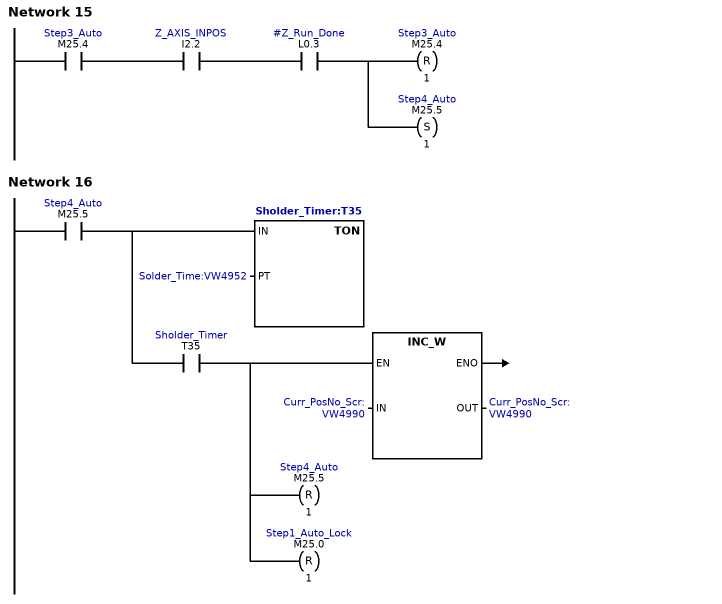
[picture p24: SBR34 networks 15-16]
Network 15
LD     Step3_Auto:M25.4
A      Z_AXIS_INPOS:I2.2
A      #Z_Run_Done:L0.3
R      Step3_Auto:M25.4, 1
S      Step4_Auto:M25.5, 1
Network 16
LD     Step4_Auto:M25.5
TON    Sholder_Timer:T35, Solder_Time:VW4952
A      Sholder_Timer:T35
INCW   Curr_PosNo_Scr:VW4990
R      Step4_Auto:M25.5, 1
R      Step1_Auto_Lock:M25.0, 1
END_SUBROUTINE_BLOCK

SUBROUTINE_BLOCK Setting:SBR35
TITLE=子例程注释
VAR_INPUT
MainScreen:WORD;	// LW0 
END_VAR
VAR
X_Home_Err:BYTE;	// LB2 
Y_Home_Err:BYTE;	// LB3 
Z_Home_Err:BYTE;	// LB4 
X_Teach_Done:BOOL;	// L5.0 
Y_Teach_Done:BOOL;	// L5.1 
Z_Teach_Done:BOOL;	// L5.2 
Z_Up_Done:BOOL;	// L5.3 
X_JOG_ERR:BYTE;	// LB6 
Y_JOG_ERR:BYTE;	// LB7 
Z_JOG_ERR:BYTE;	// LB8 
X_Curr_Dir:BOOL;	// L9.0 
Y_Curr_Dir:BOOL;	// L9.1 
Z_Curr_Dir:BOOL;	// L9.2 
END_VAR
BEGIN
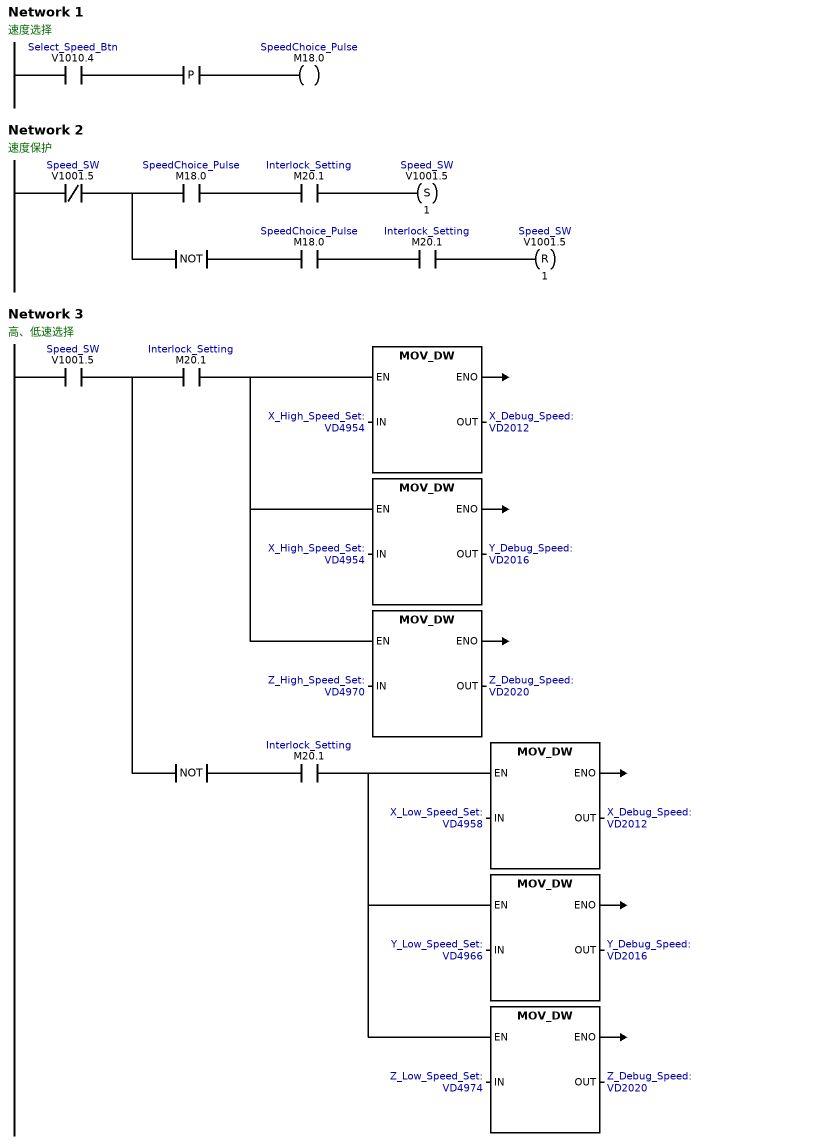
Network 1
// 速度选择
LD     Select_Speed_Btn:V1010.4
EU
=      SpeedChoice_Pulse:M18.0
Network 2
// 速度保护
LDN    Speed_SW:V1001.5
LPS
A      SpeedChoice_Pulse:M18.0
A      Interlock_Setting:M20.1
S      Speed_SW:V1001.5, 1
LPP
NOT
A      SpeedChoice_Pulse:M18.0
A      Interlock_Setting:M20.1
R      Speed_SW:V1001.5, 1
Network 3
// 高、低速选择
LD     Speed_SW:V1001.5
LPS
A      Interlock_Setting:M20.1
MOVD   X_High_Speed_Set:VD4954, X_Debug_Speed:VD2012
MOVD   X_High_Speed_Set:VD4954, Y_Debug_Speed:VD2016
MOVD   Z_High_Speed_Set:VD4970, Z_Debug_Speed:VD2020
LPP
NOT
A      Interlock_Setting:M20.1
MOVD   X_Low_Speed_Set:VD4958, X_Debug_Speed:VD2012
MOVD   Y_Low_Speed_Set:VD4966, Y_Debug_Speed:VD2016
MOVD   Z_Low_Speed_Set:VD4974, Z_Debug_Speed:VD2020
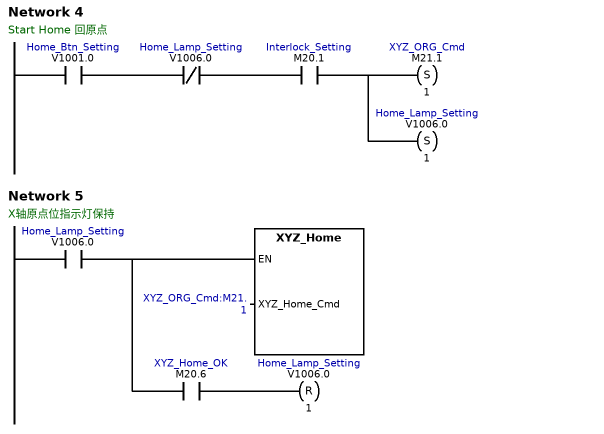
Network 4
// Start Home 回原点
LD     Home_Btn_Setting:V1001.0
AN     Home_Lamp_Setting:V1006.0
A      Interlock_Setting:M20.1
S      XYZ_ORG_Cmd:M21.1, 1
S      Home_Lamp_Setting:V1006.0, 1
Network 5
// X轴原点位指示灯保持
LD     Home_Lamp_Setting:V1006.0
CALL   XYZ_Home:SBR37, XYZ_ORG_Cmd:M21.1
A      XYZ_Home_OK:M20.6
R      Home_Lamp_Setting:V1006.0, 1
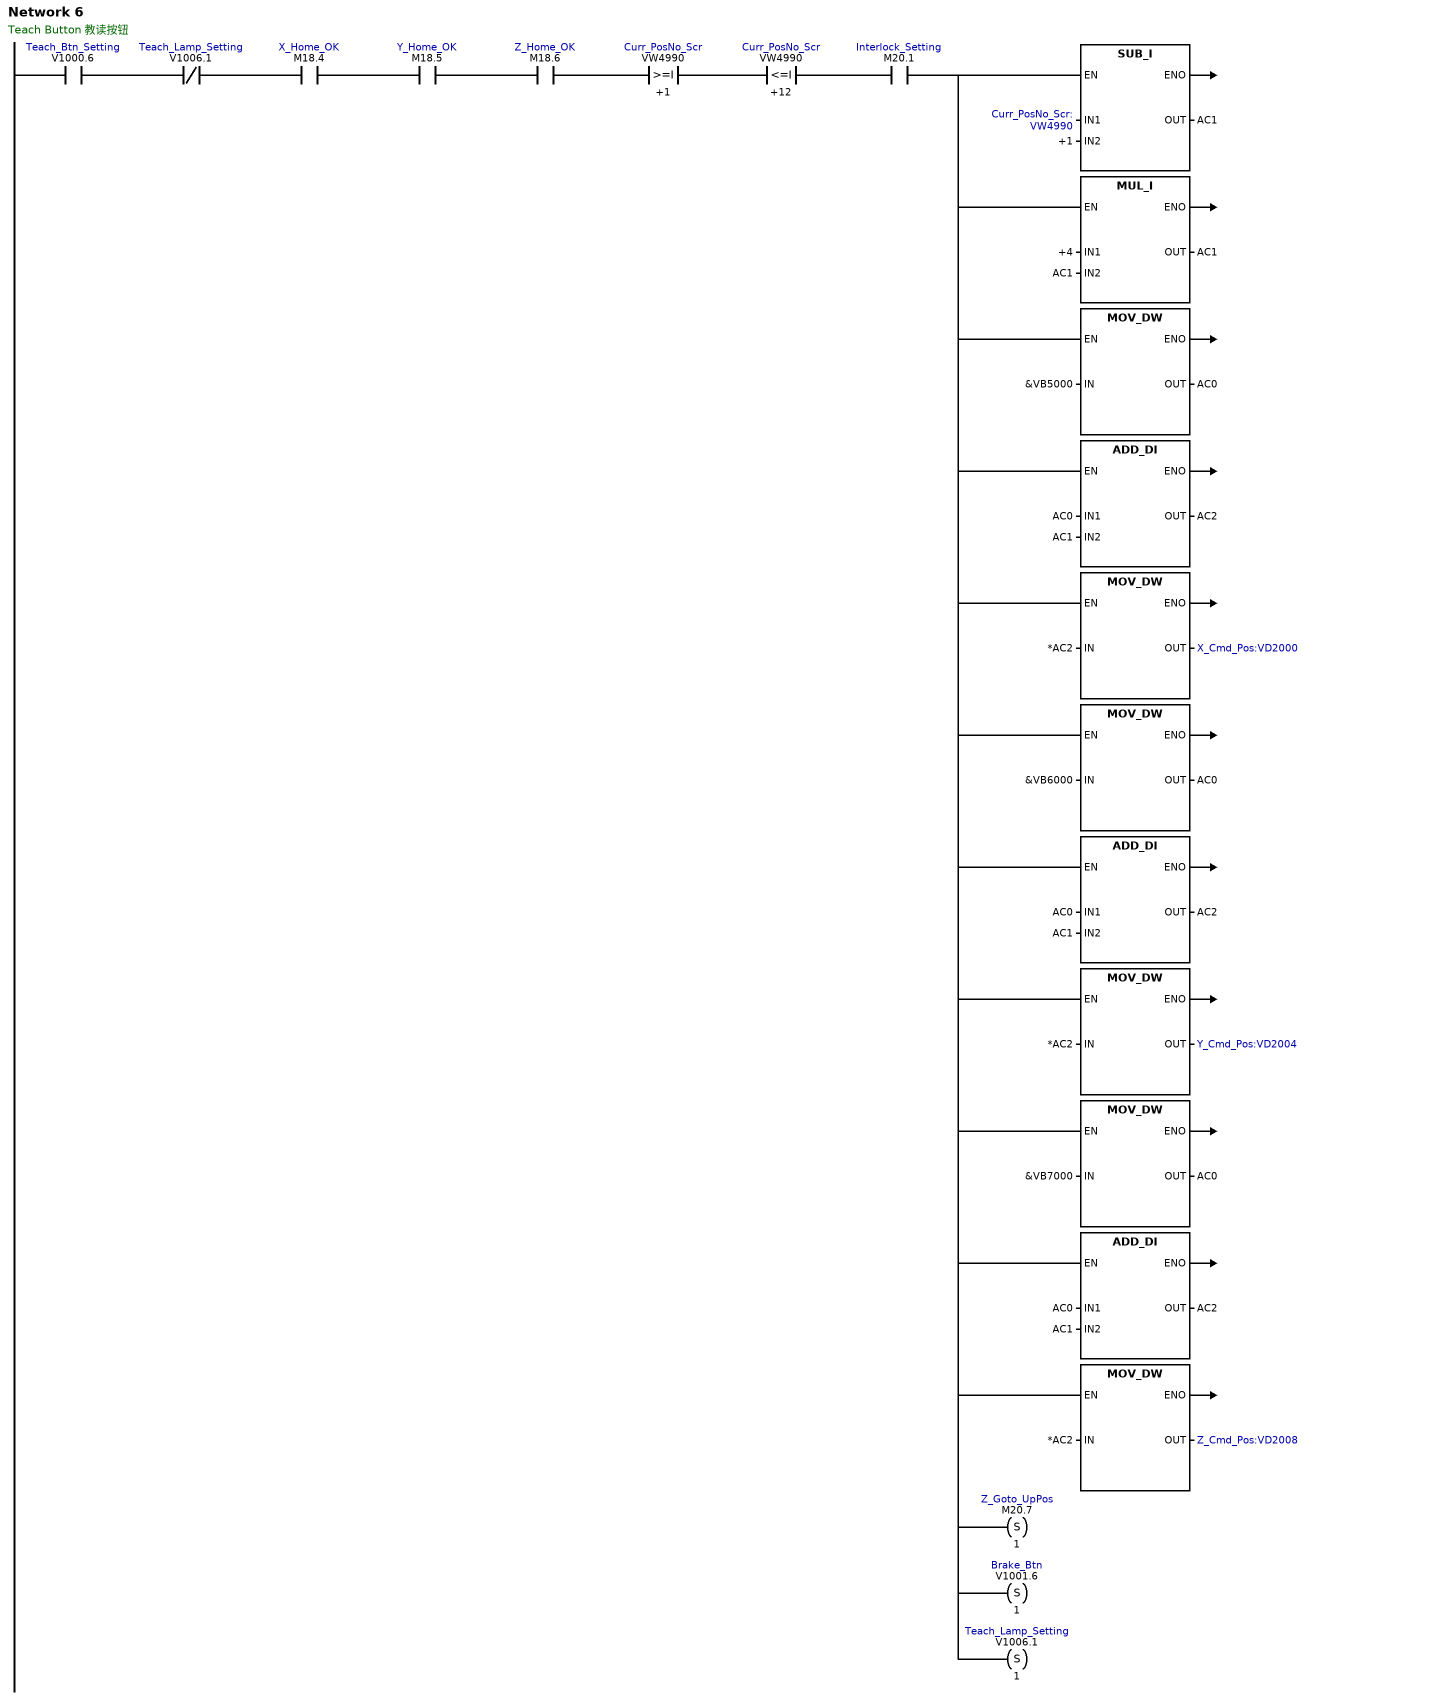
Network 6
// Teach Button 教读按钮 
LD     Teach_Btn_Setting:V1000.6
AN     Teach_Lamp_Setting:V1006.1
A      X_Home_OK:M18.4
A      Y_Home_OK:M18.5
A      Z_Home_OK:M18.6
AW>=   Curr_PosNo_Scr:VW4990, +1
AW<=   Curr_PosNo_Scr:VW4990, +12
A      Interlock_Setting:M20.1
MOVW   Curr_PosNo_Scr:VW4990, AC1
-I     +1, AC1
*I     +4, AC1
MOVD   &VB5000, AC0
MOVD   AC0, AC2
+D     AC1, AC2
MOVD   *AC2, X_Cmd_Pos:VD2000
MOVD   &VB6000, AC0
MOVD   AC0, AC2
+D     AC1, AC2
MOVD   *AC2, Y_Cmd_Pos:VD2004
MOVD   &VB7000, AC0
MOVD   AC0, AC2
+D     AC1, AC2
MOVD   *AC2, Z_Cmd_Pos:VD2008
S      Z_Goto_UpPos:M20.7, 1
S      Brake_Btn:V1001.6, 1
S      Teach_Lamp_Setting:V1006.1, 1
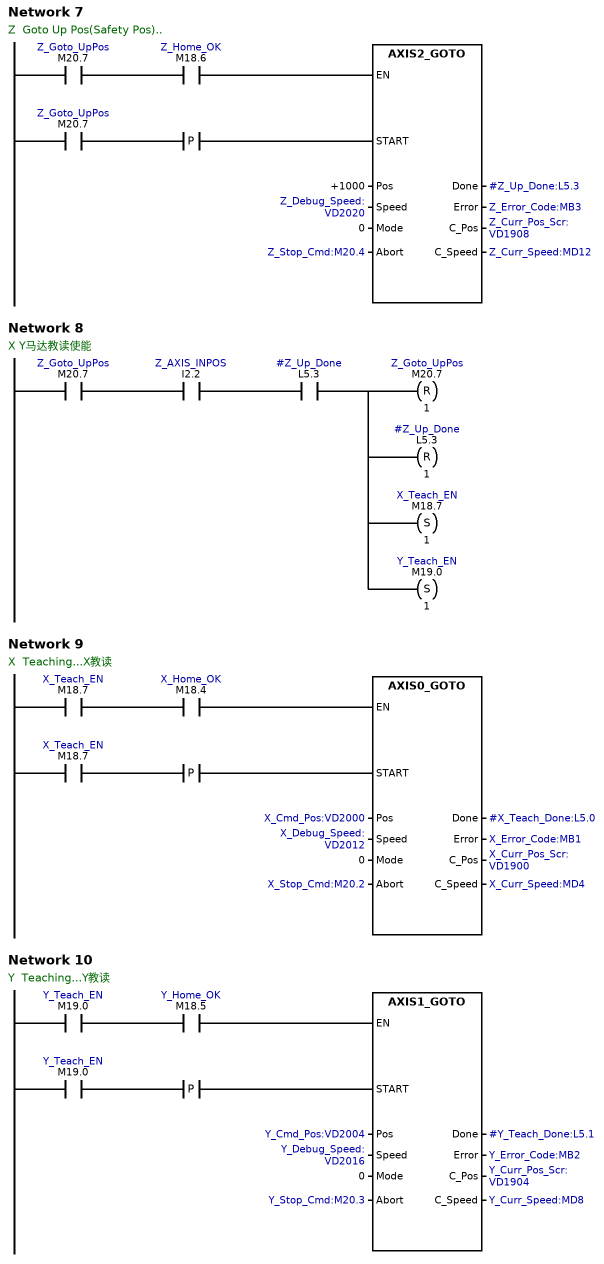
Network 7
// Z  Goto Up Pos(Safety Pos)..
LD     Z_Goto_UpPos:M20.7
A      Z_Home_OK:M18.6
=      L60.0
LD     Z_Goto_UpPos:M20.7
EU
=      L63.7
LD     L60.0
CALL   AXIS2_GOTO:SBR25, L63.7, +1000, Z_Debug_Speed:VD2020, 0, Z_Stop_Cmd:M20.4, #Z_Up_Done:L5.3, Z_Error_Code:MB3, Z_Curr_Pos_Scr:VD1908, Z_Curr_Speed:MD12
Network 8
// X Y马达教读使能
LD     Z_Goto_UpPos:M20.7
A      Z_AXIS_INPOS:I2.2
A      #Z_Up_Done:L5.3
R      Z_Goto_UpPos:M20.7, 1
R      #Z_Up_Done:L5.3, 1
S      X_Teach_EN:M18.7, 1
S      Y_Teach_EN:M19.0, 1
Network 9
// X  Teaching...X教读
LD     X_Teach_EN:M18.7
A      X_Home_OK:M18.4
=      L60.0
LD     X_Teach_EN:M18.7
EU
=      L63.7
LD     L60.0
CALL   AXIS0_GOTO:SBR3, L63.7, X_Cmd_Pos:VD2000, X_Debug_Speed:VD2012, 0, X_Stop_Cmd:M20.2, #X_Teach_Done:L5.0, X_Error_Code:MB1, X_Curr_Pos_Scr:VD1900, X_Curr_Speed:MD4
Network 10
// Y  Teaching...Y教读
LD     Y_Teach_EN:M19.0
A      Y_Home_OK:M18.5
=      L60.0
LD     Y_Teach_EN:M19.0
EU
=      L63.7
LD     L60.0
CALL   AXIS1_GOTO:SBR14, L63.7, Y_Cmd_Pos:VD2004, Y_Debug_Speed:VD2016, 0, Y_Stop_Cmd:M20.3, #Y_Teach_Done:L5.1, Y_Error_Code:MB2, Y_Curr_Pos_Scr:VD1904, Y_Curr_Speed:MD8
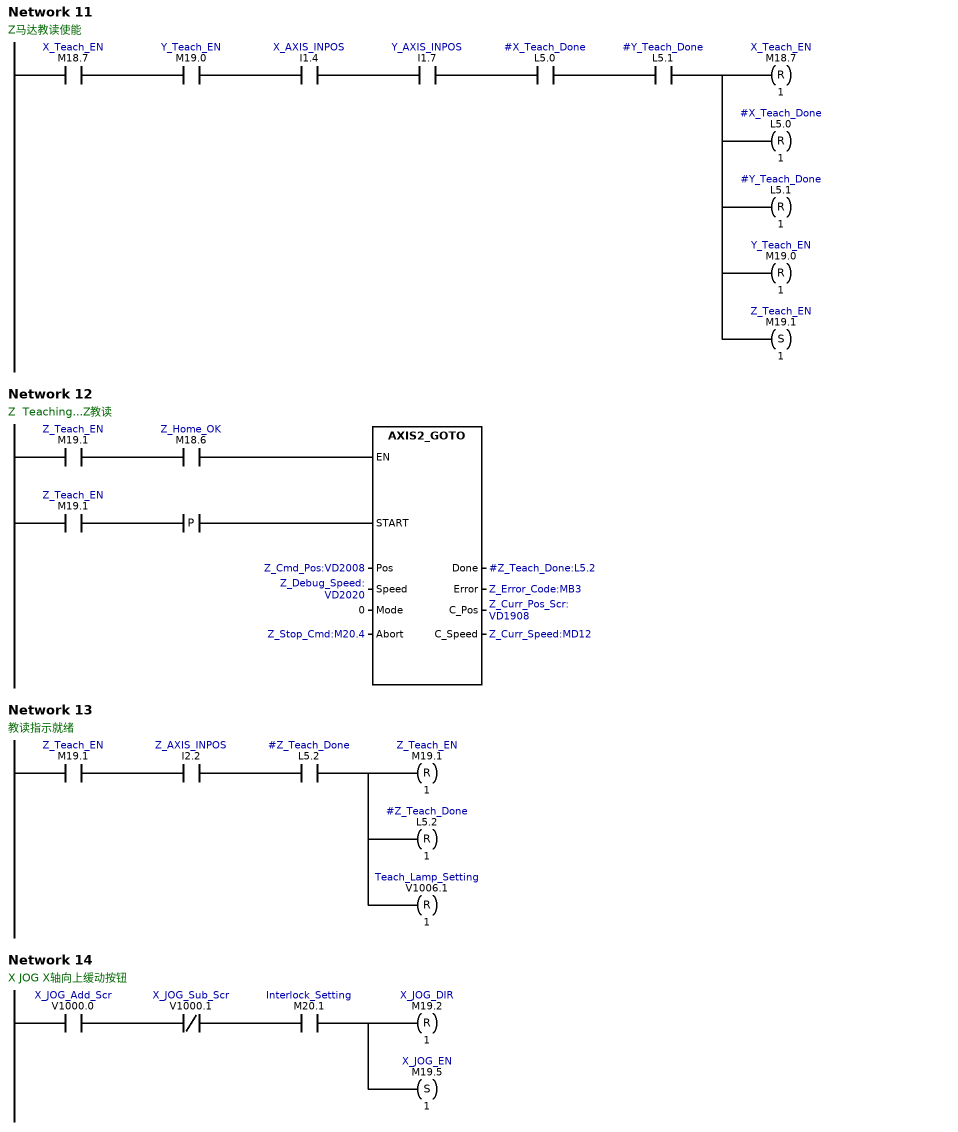
Network 11
// Z马达教读使能
LD     X_Teach_EN:M18.7
A      Y_Teach_EN:M19.0
A      X_AXIS_INPOS:I1.4
A      Y_AXIS_INPOS:I1.7
A      #X_Teach_Done:L5.0
A      #Y_Teach_Done:L5.1
R      X_Teach_EN:M18.7, 1
R      #X_Teach_Done:L5.0, 1
R      #Y_Teach_Done:L5.1, 1
R      Y_Teach_EN:M19.0, 1
S      Z_Teach_EN:M19.1, 1
Network 12
// Z  Teaching...Z教读
LD     Z_Teach_EN:M19.1
A      Z_Home_OK:M18.6
=      L60.0
LD     Z_Teach_EN:M19.1
EU
=      L63.7
LD     L60.0
CALL   AXIS2_GOTO:SBR25, L63.7, Z_Cmd_Pos:VD2008, Z_Debug_Speed:VD2020, 0, Z_Stop_Cmd:M20.4, #Z_Teach_Done:L5.2, Z_Error_Code:MB3, Z_Curr_Pos_Scr:VD1908, Z_Curr_Speed:MD12
Network 13
// 教读指示就绪
LD     Z_Teach_EN:M19.1
A      Z_AXIS_INPOS:I2.2
A      #Z_Teach_Done:L5.2
R      Z_Teach_EN:M19.1, 1
R      #Z_Teach_Done:L5.2, 1
R      Teach_Lamp_Setting:V1006.1, 1
Network 14
// X JOG X轴向上缓动按钮
LD     X_JOG_Add_Scr:V1000.0
AN     X_JOG_Sub_Scr:V1000.1
A      Interlock_Setting:M20.1
R      X_JOG_DIR:M19.2, 1
S      X_JOG_EN:M19.5, 1
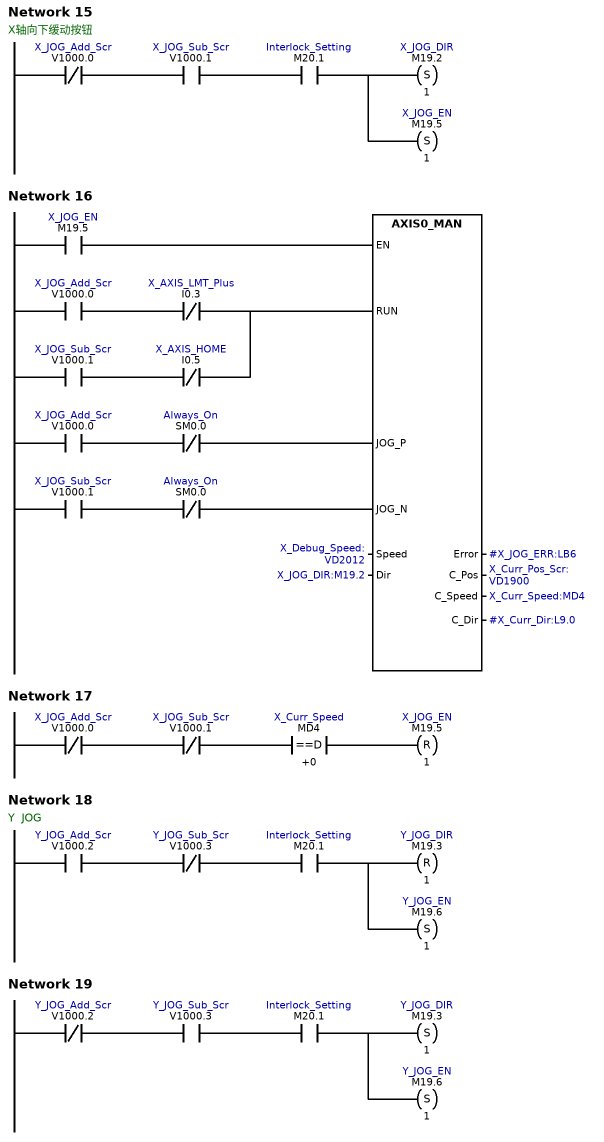
Network 15
// X轴向下缓动按钮
LDN    X_JOG_Add_Scr:V1000.0
A      X_JOG_Sub_Scr:V1000.1
A      Interlock_Setting:M20.1
S      X_JOG_DIR:M19.2, 1
S      X_JOG_EN:M19.5, 1
Network 16
LD     X_JOG_EN:M19.5
=      L60.0
LD     X_JOG_Add_Scr:V1000.0
AN     X_AXIS_LMT_Plus:I0.3
LD     X_JOG_Sub_Scr:V1000.1
AN     X_AXIS_HOME:I0.5
OLD
=      L63.7
LD     X_JOG_Add_Scr:V1000.0
AN     Always_On:SM0.0
=      L63.6
LD     X_JOG_Sub_Scr:V1000.1
AN     Always_On:SM0.0
=      L63.5
LD     L60.0
CALL   AXIS0_MAN:SBR2, L63.7, L63.6, L63.5, X_Debug_Speed:VD2012, X_JOG_DIR:M19.2, #X_JOG_ERR:LB6, X_Curr_Pos_Scr:VD1900, X_Curr_Speed:MD4, #X_Curr_Dir:L9.0
Network 17
LDN    X_JOG_Add_Scr:V1000.0
AN     X_JOG_Sub_Scr:V1000.1
AD=    X_Curr_Speed:MD4, +0
R      X_JOG_EN:M19.5, 1
Network 18
// Y  JOG
LD     Y_JOG_Add_Scr:V1000.2
AN     Y_JOG_Sub_Scr:V1000.3
A      Interlock_Setting:M20.1
R      Y_JOG_DIR:M19.3, 1
S      Y_JOG_EN:M19.6, 1
Network 19
LDN    Y_JOG_Add_Scr:V1000.2
A      Y_JOG_Sub_Scr:V1000.3
A      Interlock_Setting:M20.1
S      Y_JOG_DIR:M19.3, 1
S      Y_JOG_EN:M19.6, 1
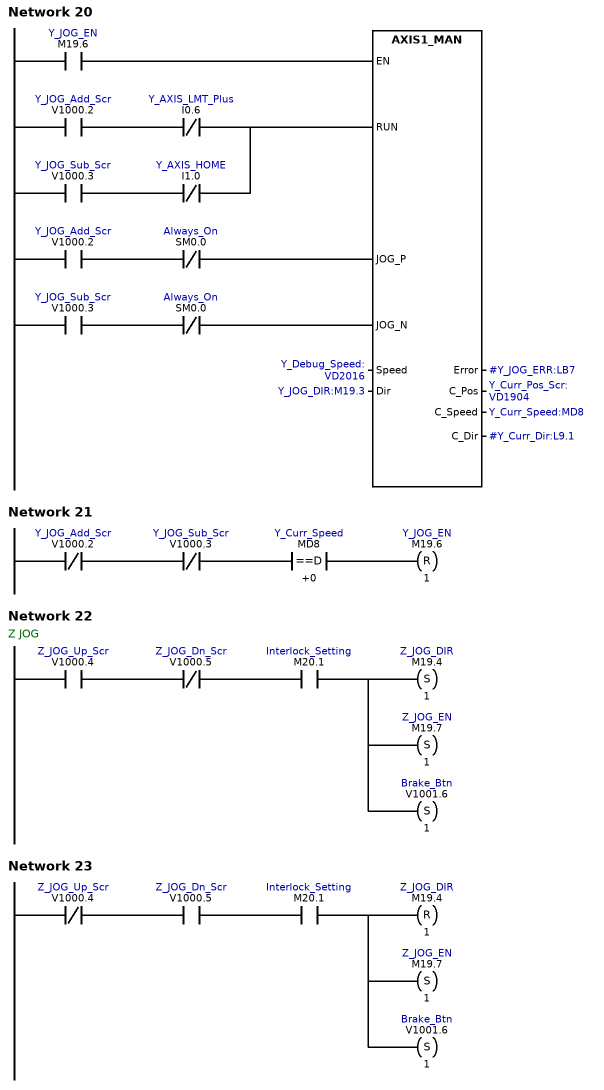
Network 20
LD     Y_JOG_EN:M19.6
=      L60.0
LD     Y_JOG_Add_Scr:V1000.2
AN     Y_AXIS_LMT_Plus:I0.6
LD     Y_JOG_Sub_Scr:V1000.3
AN     Y_AXIS_HOME:I1.0
OLD
=      L63.7
LD     Y_JOG_Add_Scr:V1000.2
AN     Always_On:SM0.0
=      L63.6
LD     Y_JOG_Sub_Scr:V1000.3
AN     Always_On:SM0.0
=      L63.5
LD     L60.0
CALL   AXIS1_MAN:SBR13, L63.7, L63.6, L63.5, Y_Debug_Speed:VD2016, Y_JOG_DIR:M19.3, #Y_JOG_ERR:LB7, Y_Curr_Pos_Scr:VD1904, Y_Curr_Speed:MD8, #Y_Curr_Dir:L9.1
Network 21
LDN    Y_JOG_Add_Scr:V1000.2
AN     Y_JOG_Sub_Scr:V1000.3
AD=    Y_Curr_Speed:MD8, +0
R      Y_JOG_EN:M19.6, 1
Network 22
// Z JOG
LD     Z_JOG_Up_Scr:V1000.4
AN     Z_JOG_Dn_Scr:V1000.5
A      Interlock_Setting:M20.1
S      Z_JOG_DIR:M19.4, 1
S      Z_JOG_EN:M19.7, 1
S      Brake_Btn:V1001.6, 1
Network 23
LDN    Z_JOG_Up_Scr:V1000.4
A      Z_JOG_Dn_Scr:V1000.5
A      Interlock_Setting:M20.1
R      Z_JOG_DIR:M19.4, 1
S      Z_JOG_EN:M19.7, 1
S      Brake_Btn:V1001.6, 1
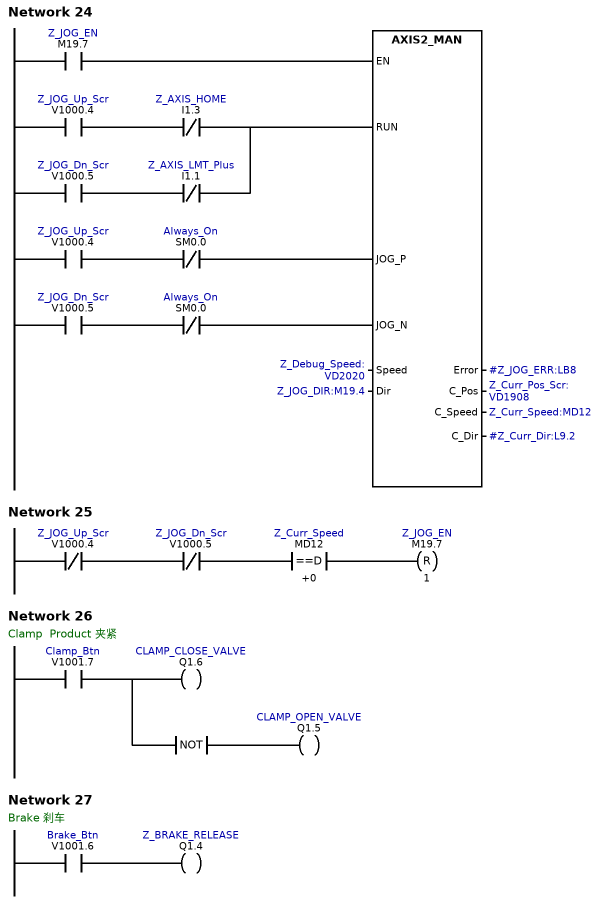
Network 24
LD     Z_JOG_EN:M19.7
=      L60.0
LD     Z_JOG_Up_Scr:V1000.4
AN     Z_AXIS_HOME:I1.3
LD     Z_JOG_Dn_Scr:V1000.5
AN     Z_AXIS_LMT_Plus:I1.1
OLD
=      L63.7
LD     Z_JOG_Up_Scr:V1000.4
AN     Always_On:SM0.0
=      L63.6
LD     Z_JOG_Dn_Scr:V1000.5
AN     Always_On:SM0.0
=      L63.5
LD     L60.0
CALL   AXIS2_MAN:SBR24, L63.7, L63.6, L63.5, Z_Debug_Speed:VD2020, Z_JOG_DIR:M19.4, #Z_JOG_ERR:LB8, Z_Curr_Pos_Scr:VD1908, Z_Curr_Speed:MD12, #Z_Curr_Dir:L9.2
Network 25
LDN    Z_JOG_Up_Scr:V1000.4
AN     Z_JOG_Dn_Scr:V1000.5
AD=    Z_Curr_Speed:MD12, +0
R      Z_JOG_EN:M19.7, 1
Network 26
// Clamp  Product 夹紧
LD     Clamp_Btn:V1001.7
=      CLAMP_CLOSE_VALVE:Q1.6
NOT
=      CLAMP_OPEN_VALVE:Q1.5
Network 27
// Brake 刹车
LD     Brake_Btn:V1001.6
=      Z_BRAKE_RELEASE:Q1.4
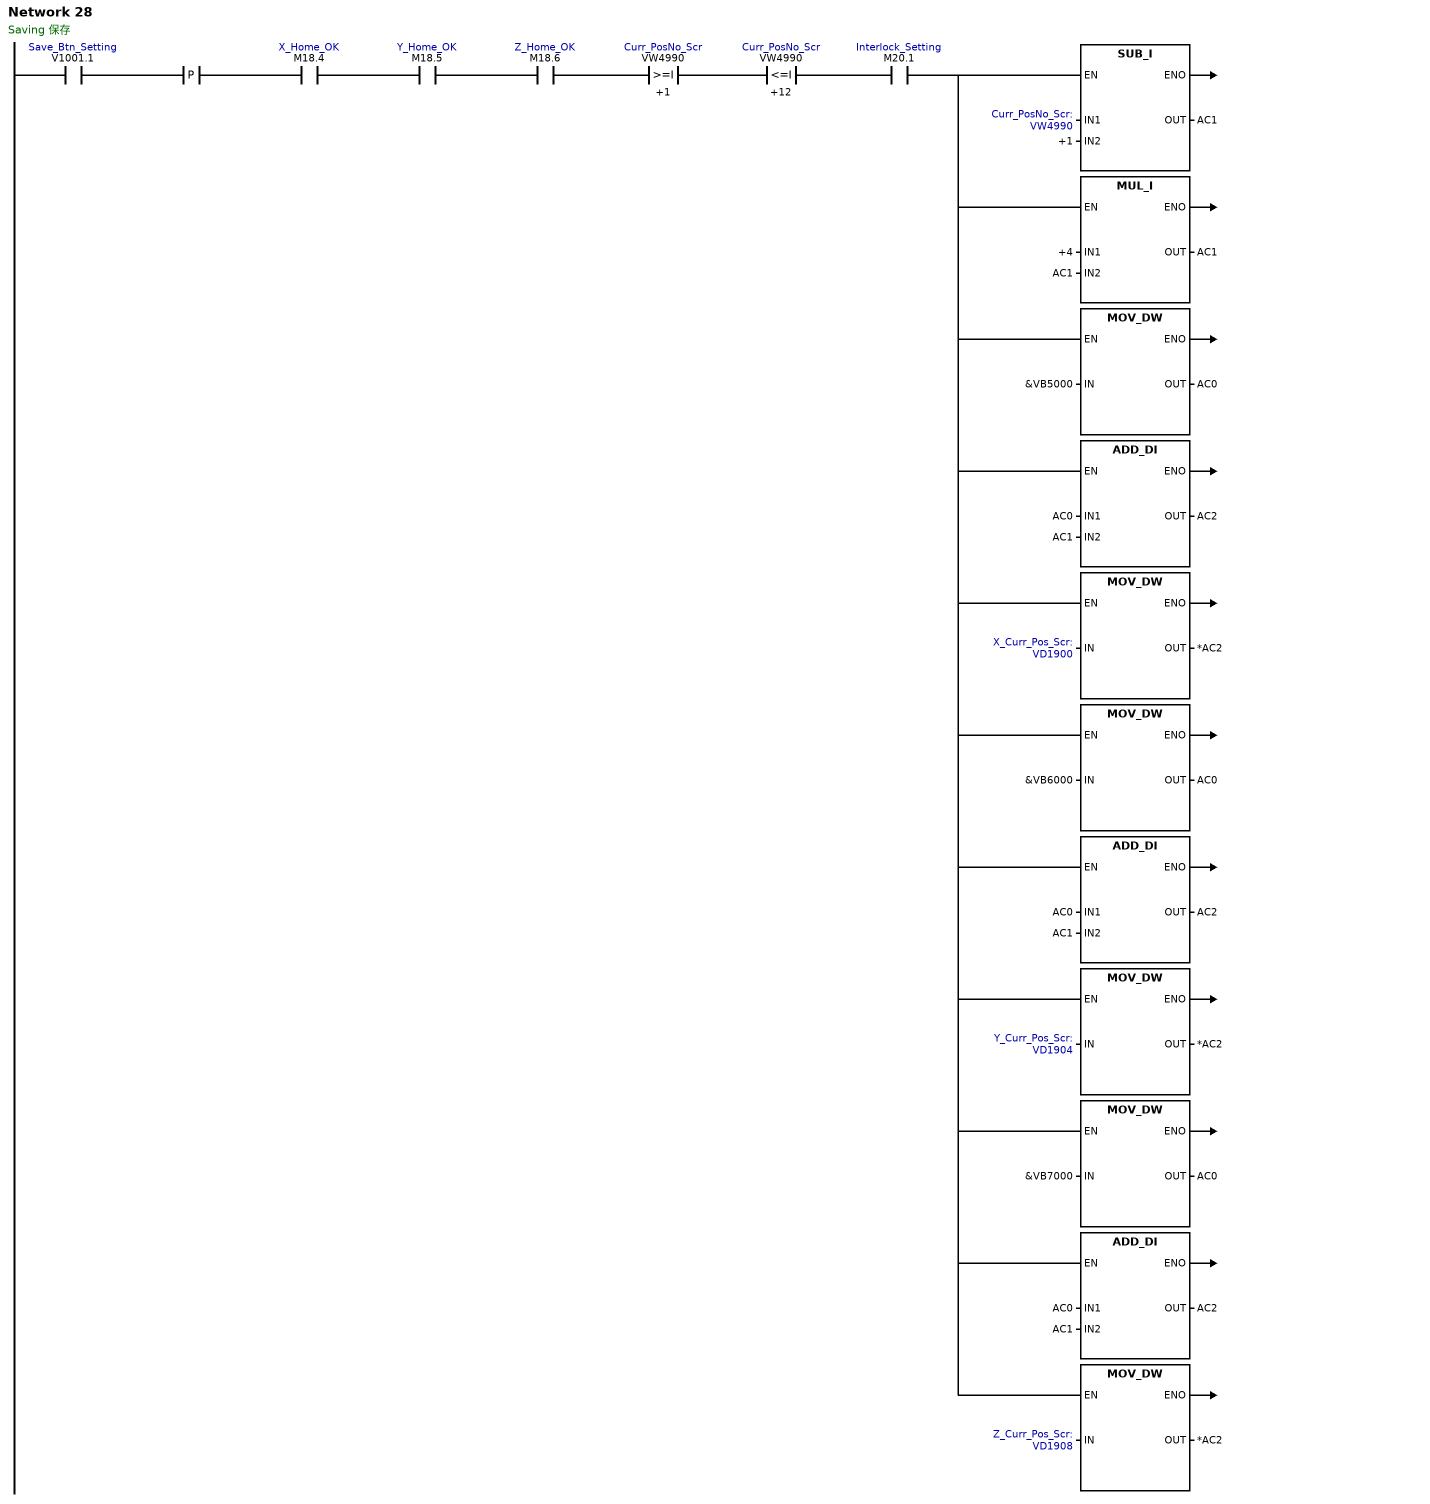
Network 28
// Saving 保存
LD     Save_Btn_Setting:V1001.1
EU
A      X_Home_OK:M18.4
A      Y_Home_OK:M18.5
A      Z_Home_OK:M18.6
AW>=   Curr_PosNo_Scr:VW4990, +1
AW<=   Curr_PosNo_Scr:VW4990, +12
A      Interlock_Setting:M20.1
MOVW   Curr_PosNo_Scr:VW4990, AC1
-I     +1, AC1
*I     +4, AC1
MOVD   &VB5000, AC0
MOVD   AC0, AC2
+D     AC1, AC2
MOVD   X_Curr_Pos_Scr:VD1900, *AC2
MOVD   &VB6000, AC0
MOVD   AC0, AC2
+D     AC1, AC2
MOVD   Y_Curr_Pos_Scr:VD1904, *AC2
MOVD   &VB7000, AC0
MOVD   AC0, AC2
+D     AC1, AC2
MOVD   Z_Curr_Pos_Scr:VD1908, *AC2
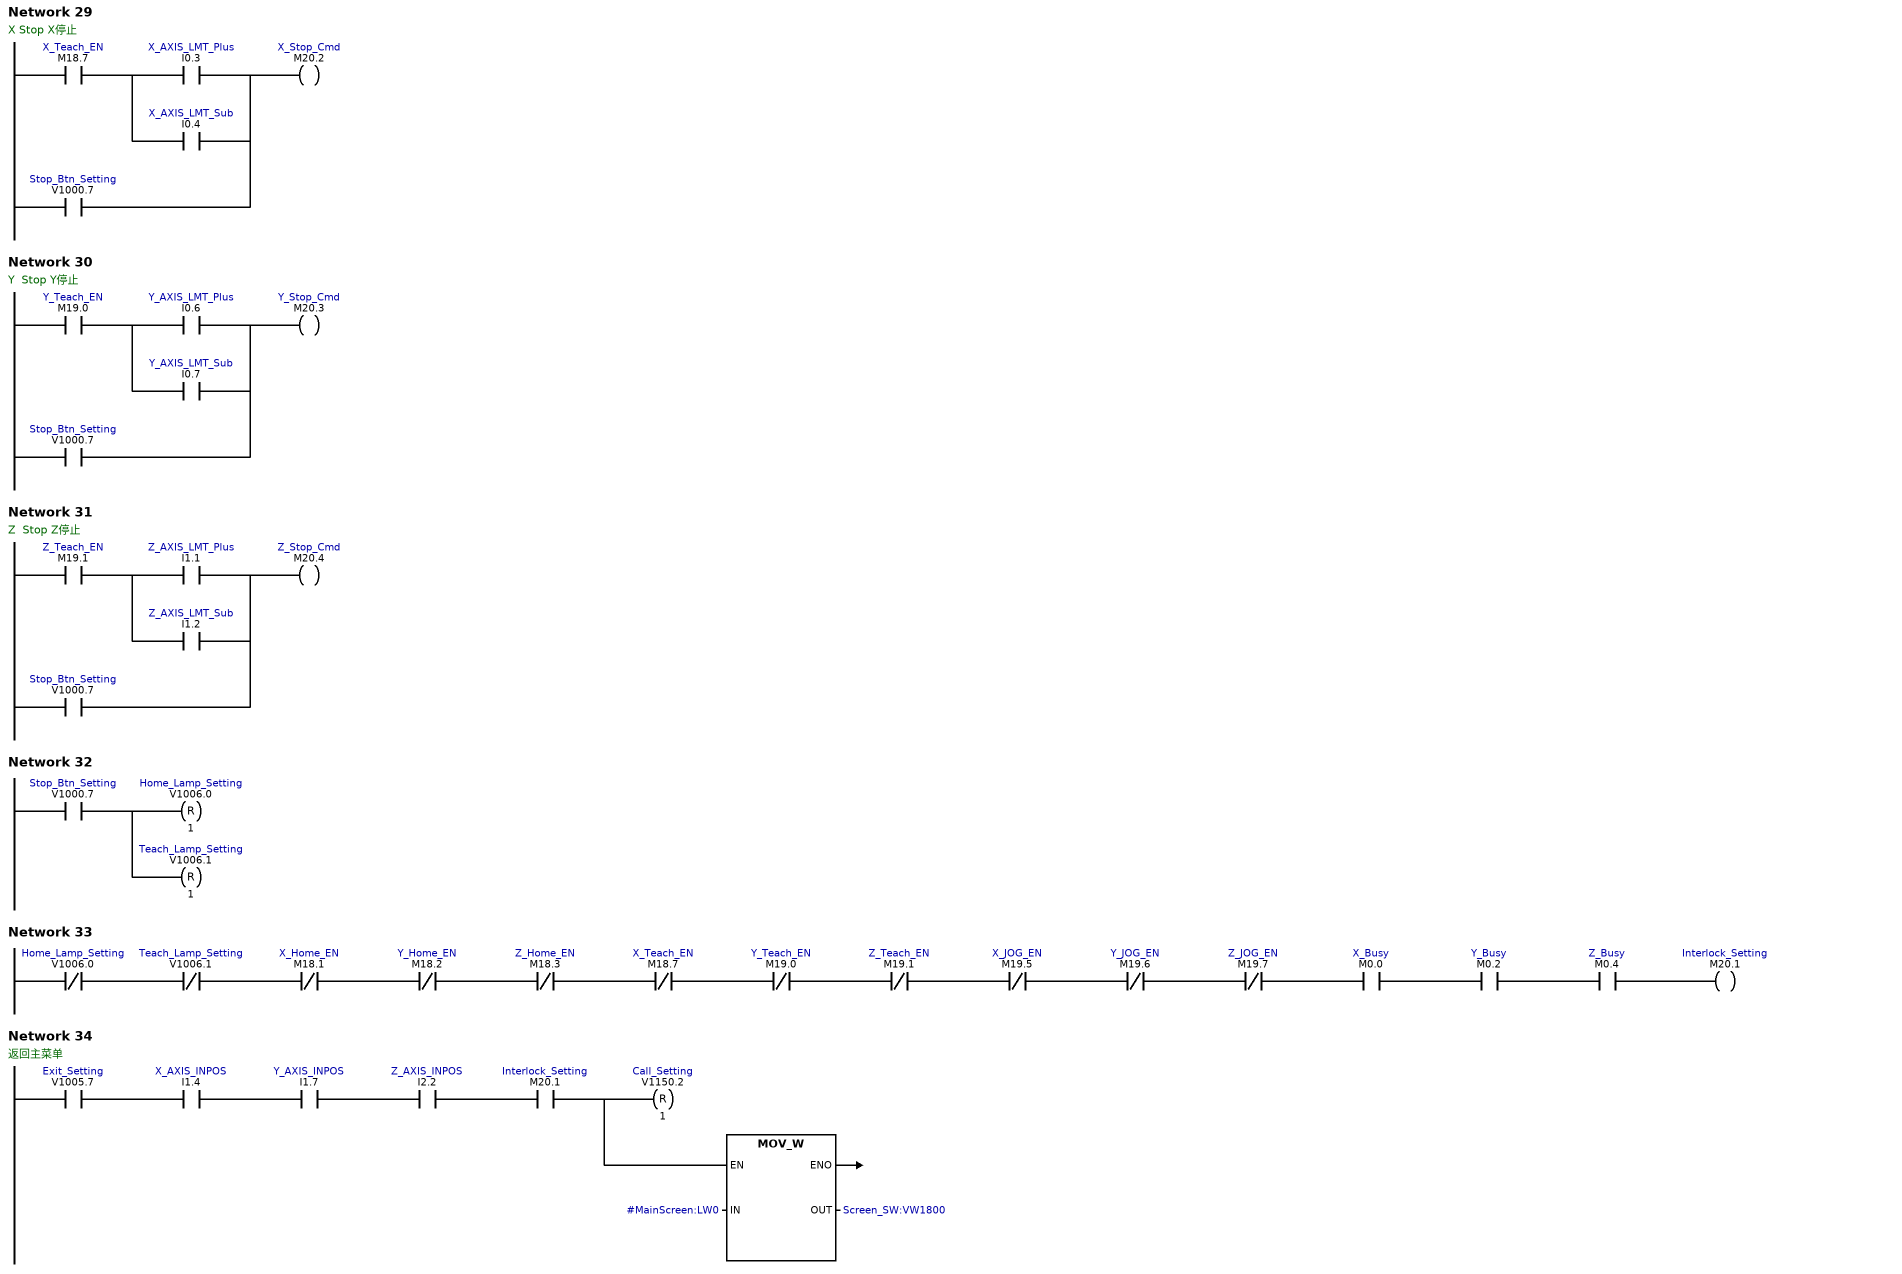
Network 29
// X Stop X停止
LD     X_Teach_EN:M18.7
LD     X_AXIS_LMT_Plus:I0.3
O      X_AXIS_LMT_Sub:I0.4
ALD
O      Stop_Btn_Setting:V1000.7
=      X_Stop_Cmd:M20.2
Network 30
// Y  Stop Y停止
LD     Y_Teach_EN:M19.0
LD     Y_AXIS_LMT_Plus:I0.6
O      Y_AXIS_LMT_Sub:I0.7
ALD
O      Stop_Btn_Setting:V1000.7
=      Y_Stop_Cmd:M20.3
Network 31
// Z  Stop Z停止
LD     Z_Teach_EN:M19.1
LD     Z_AXIS_LMT_Plus:I1.1
O      Z_AXIS_LMT_Sub:I1.2
ALD
O      Stop_Btn_Setting:V1000.7
=      Z_Stop_Cmd:M20.4
Network 32
LD     Stop_Btn_Setting:V1000.7
R      Home_Lamp_Setting:V1006.0, 1
R      Teach_Lamp_Setting:V1006.1, 1
Network 33
LDN    Home_Lamp_Setting:V1006.0
AN     Teach_Lamp_Setting:V1006.1
AN     X_Home_EN:M18.1
AN     Y_Home_EN:M18.2
AN     Z_Home_EN:M18.3
AN     X_Teach_EN:M18.7
AN     Y_Teach_EN:M19.0
AN     Z_Teach_EN:M19.1
AN     X_JOG_EN:M19.5
AN     Y_JOG_EN:M19.6
AN     Z_JOG_EN:M19.7
A      X_Busy:M0.0
A      Y_Busy:M0.2
A      Z_Busy:M0.4
=      Interlock_Setting:M20.1
Network 34
// 返回主菜单
LD     Exit_Setting:V1005.7
A      X_AXIS_INPOS:I1.4
A      Y_AXIS_INPOS:I1.7
A      Z_AXIS_INPOS:I2.2
A      Interlock_Setting:M20.1
R      Call_Setting:V1150.2, 1
MOVW   #MainScreen:LW0, Screen_SW:VW1800
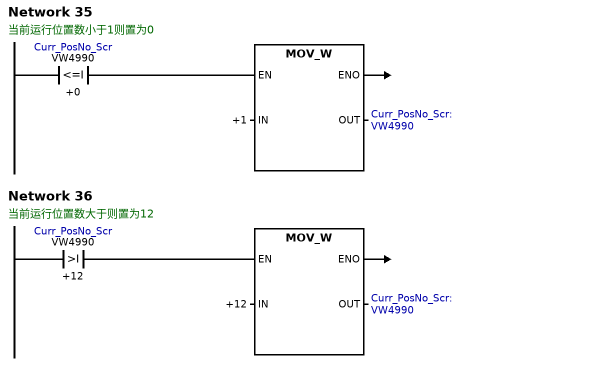
Network 35
// 当前运行位置数小于1则置为0
LDW<=  Curr_PosNo_Scr:VW4990, +0
MOVW   +1, Curr_PosNo_Scr:VW4990
Network 36
// 当前运行位置数大于则置为12
LDW>   Curr_PosNo_Scr:VW4990, +12
MOVW   +12, Curr_PosNo_Scr:VW4990
END_SUBROUTINE_BLOCK

SUBROUTINE_BLOCK Alarm_Process:SBR36
TITLE=子例程注释
BEGIN
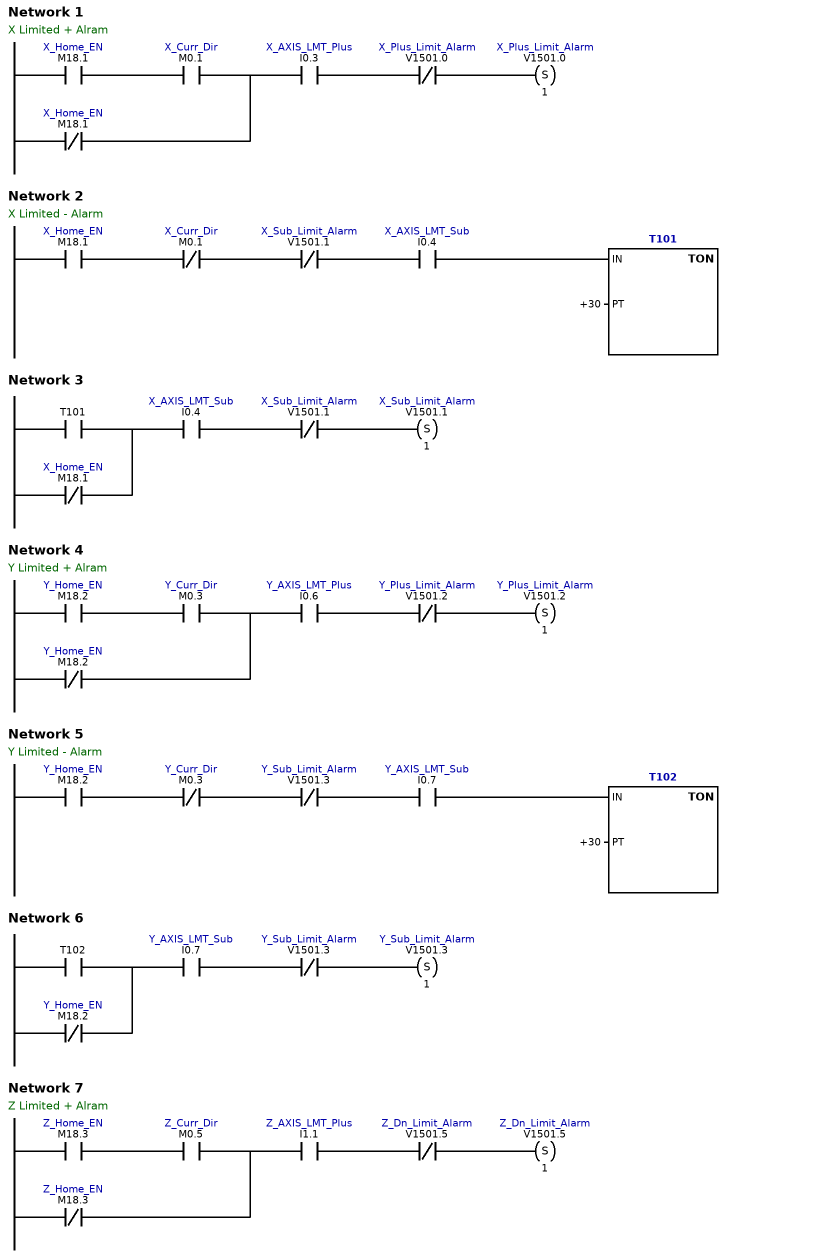
Network 1
// X Limited + Alram
LD     X_Home_EN:M18.1
A      X_Curr_Dir:M0.1
ON     X_Home_EN:M18.1
A      X_AXIS_LMT_Plus:I0.3
AN     X_Plus_Limit_Alarm:V1501.0
S      X_Plus_Limit_Alarm:V1501.0, 1
Network 2
// X Limited - Alarm
LD     X_Home_EN:M18.1
AN     X_Curr_Dir:M0.1
AN     X_Sub_Limit_Alarm:V1501.1
A      X_AXIS_LMT_Sub:I0.4
TON    T101, +30
Network 3
LD     T101
ON     X_Home_EN:M18.1
A      X_AXIS_LMT_Sub:I0.4
AN     X_Sub_Limit_Alarm:V1501.1
S      X_Sub_Limit_Alarm:V1501.1, 1
Network 4
// Y Limited + Alram
LD     Y_Home_EN:M18.2
A      Y_Curr_Dir:M0.3
ON     Y_Home_EN:M18.2
A      Y_AXIS_LMT_Plus:I0.6
AN     Y_Plus_Limit_Alarm:V1501.2
S      Y_Plus_Limit_Alarm:V1501.2, 1
Network 5
// Y Limited - Alarm
LD     Y_Home_EN:M18.2
AN     Y_Curr_Dir:M0.3
AN     Y_Sub_Limit_Alarm:V1501.3
A      Y_AXIS_LMT_Sub:I0.7
TON    T102, +30
Network 6
LD     T102
ON     Y_Home_EN:M18.2
A      Y_AXIS_LMT_Sub:I0.7
AN     Y_Sub_Limit_Alarm:V1501.3
S      Y_Sub_Limit_Alarm:V1501.3, 1
Network 7
// Z Limited + Alram
LD     Z_Home_EN:M18.3
A      Z_Curr_Dir:M0.5
ON     Z_Home_EN:M18.3
A      Z_AXIS_LMT_Plus:I1.1
AN     Z_Dn_Limit_Alarm:V1501.5
S      Z_Dn_Limit_Alarm:V1501.5, 1
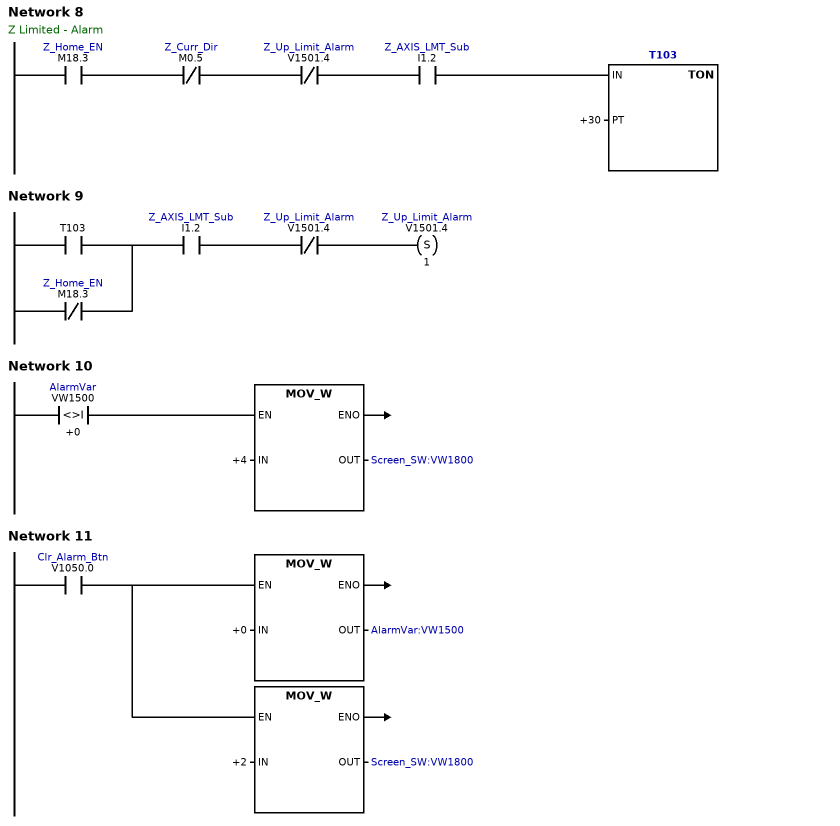
Network 8
// Z Limited - Alarm
LD     Z_Home_EN:M18.3
AN     Z_Curr_Dir:M0.5
AN     Z_Up_Limit_Alarm:V1501.4
A      Z_AXIS_LMT_Sub:I1.2
TON    T103, +30
Network 9
LD     T103
ON     Z_Home_EN:M18.3
A      Z_AXIS_LMT_Sub:I1.2
AN     Z_Up_Limit_Alarm:V1501.4
S      Z_Up_Limit_Alarm:V1501.4, 1
Network 10
LDW<>  AlarmVar:VW1500, +0
MOVW   +4, Screen_SW:VW1800
Network 11
LD     Clr_Alarm_Btn:V1050.0
MOVW   +0, AlarmVar:VW1500
MOVW   +2, Screen_SW:VW1800
END_SUBROUTINE_BLOCK

SUBROUTINE_BLOCK XYZ_Home:SBR37
TITLE=子例程注释
VAR_IN_OUT
XYZ_Home_Cmd:BOOL;	// L0.0 
END_VAR
BEGIN
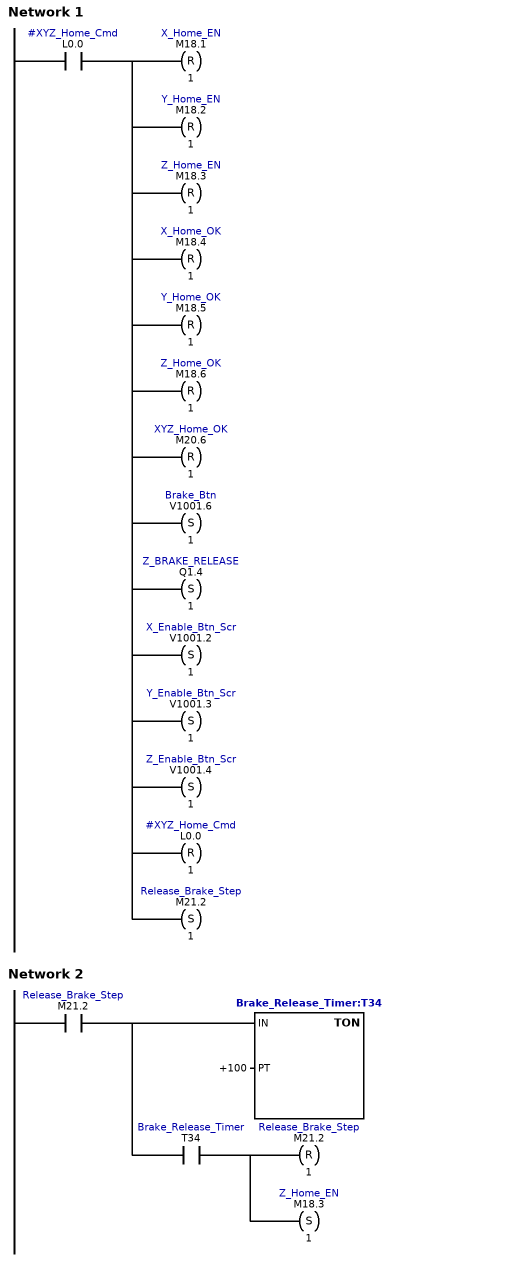
Network 1
LD     #XYZ_Home_Cmd:L0.0
R      X_Home_EN:M18.1, 1
R      Y_Home_EN:M18.2, 1
R      Z_Home_EN:M18.3, 1
R      X_Home_OK:M18.4, 1
R      Y_Home_OK:M18.5, 1
R      Z_Home_OK:M18.6, 1
R      XYZ_Home_OK:M20.6, 1
S      Brake_Btn:V1001.6, 1
S      Z_BRAKE_RELEASE:Q1.4, 1
S      X_Enable_Btn_Scr:V1001.2, 1
S      Y_Enable_Btn_Scr:V1001.3, 1
S      Z_Enable_Btn_Scr:V1001.4, 1
R      #XYZ_Home_Cmd:L0.0, 1
S      Release_Brake_Step:M21.2, 1
Network 2
LD     Release_Brake_Step:M21.2
TON    Brake_Release_Timer:T34, +100
A      Brake_Release_Timer:T34
R      Release_Brake_Step:M21.2, 1
S      Z_Home_EN:M18.3, 1
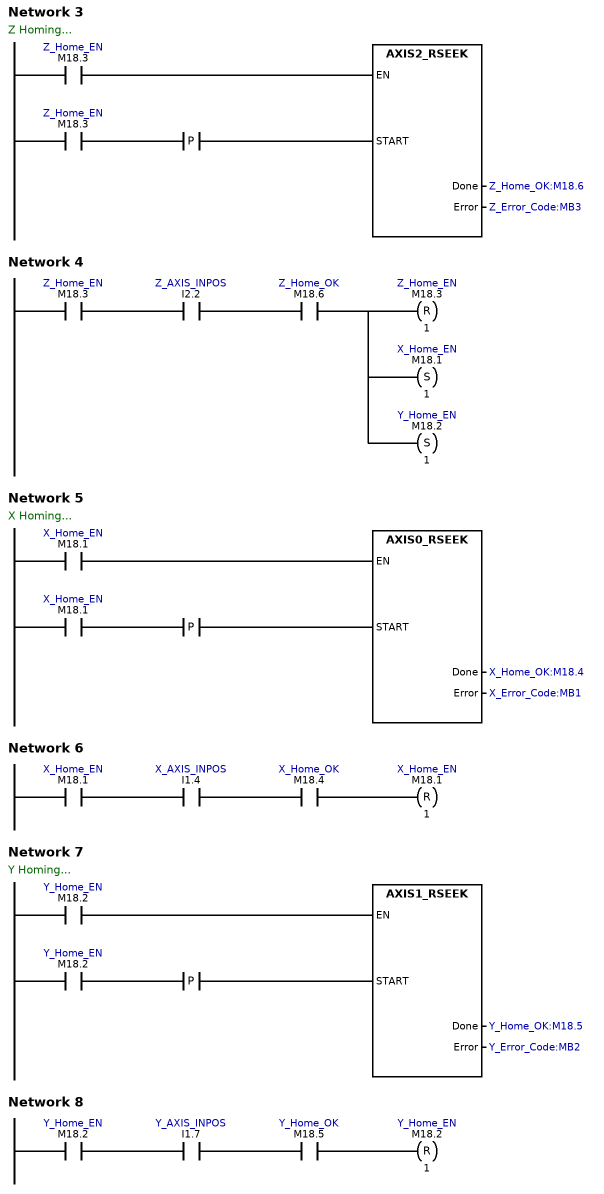
Network 3
// Z Homing...
LD     Z_Home_EN:M18.3
=      L60.0
LD     Z_Home_EN:M18.3
EU
=      L63.7
LD     L60.0
CALL   AXIS2_RSEEK:SBR27, L63.7, Z_Home_OK:M18.6, Z_Error_Code:MB3
Network 4
LD     Z_Home_EN:M18.3
A      Z_AXIS_INPOS:I2.2
A      Z_Home_OK:M18.6
R      Z_Home_EN:M18.3, 1
S      X_Home_EN:M18.1, 1
S      Y_Home_EN:M18.2, 1
Network 5
// X Homing...
LD     X_Home_EN:M18.1
=      L60.0
LD     X_Home_EN:M18.1
EU
=      L63.7
LD     L60.0
CALL   AXIS0_RSEEK:SBR5, L63.7, X_Home_OK:M18.4, X_Error_Code:MB1
Network 6
LD     X_Home_EN:M18.1
A      X_AXIS_INPOS:I1.4
A      X_Home_OK:M18.4
R      X_Home_EN:M18.1, 1
Network 7
// Y Homing...
LD     Y_Home_EN:M18.2
=      L60.0
LD     Y_Home_EN:M18.2
EU
=      L63.7
LD     L60.0
CALL   AXIS1_RSEEK:SBR16, L63.7, Y_Home_OK:M18.5, Y_Error_Code:MB2
Network 8
LD     Y_Home_EN:M18.2
A      Y_AXIS_INPOS:I1.7
A      Y_Home_OK:M18.5
R      Y_Home_EN:M18.2, 1
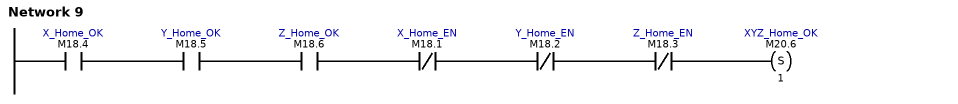
Network 9
LD     X_Home_OK:M18.4
A      Y_Home_OK:M18.5
A      Z_Home_OK:M18.6
AN     X_Home_EN:M18.1
AN     Y_Home_EN:M18.2
AN     Z_Home_EN:M18.3
S      XYZ_Home_OK:M20.6, 1
END_SUBROUTINE_BLOCK

SUBROUTINE_BLOCK solder1:SBR38
TITLE=子例程注释
VAR_IN_OUT
Solder1_Cmd:BOOL;	// L0.0 
END_VAR
VAR
Y_Run_Done:BOOL;	// L0.1 
Z_Run_Done:BOOL;	// L0.2 
X_Run_Done:BOOL;	// L0.3 
Z_Up_Done:BOOL;	// L0.4 
Z_Run_Done1:BOOL;	// L0.5 
Z_Run_Done2:BOOL;	// L0.6 
Z_Run_Done3:BOOL;	// L0.7 
X_Run_Done1:BOOL;	// L1.0 
X_Run_Done2:BOOL;	// L1.1 
Z_Run_Done4:BOOL;	// L1.2 
X_Run_Done3:BOOL;	// L1.3 
Z_Run_Done5:BOOL;	// L1.4 
END_VAR
BEGIN
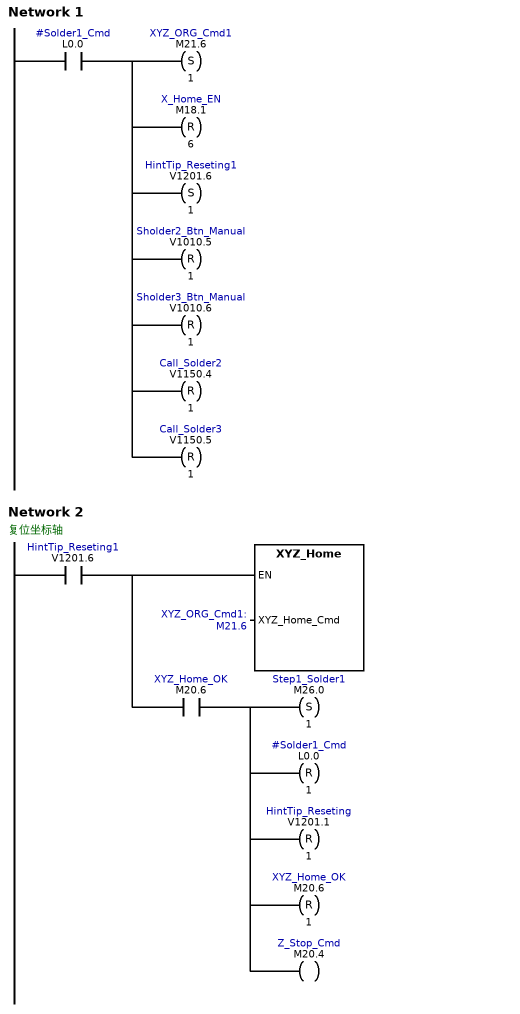
Network 1
LD     #Solder1_Cmd:L0.0
S      XYZ_ORG_Cmd1:M21.6, 1
R      X_Home_EN:M18.1, 6
S      HintTip_Reseting1:V1201.6, 1
R      Sholder2_Btn_Manual:V1010.5, 1
R      Sholder3_Btn_Manual:V1010.6, 1
R      Call_Solder2:V1150.4, 1
R      Call_Solder3:V1150.5, 1
Network 2
// 复位坐标轴
LD     HintTip_Reseting1:V1201.6
CALL   XYZ_Home:SBR37, XYZ_ORG_Cmd1:M21.6
A      XYZ_Home_OK:M20.6
S      Step1_Solder1:M26.0, 1
R      #Solder1_Cmd:L0.0, 1
R      HintTip_Reseting:V1201.1, 1
R      XYZ_Home_OK:M20.6, 1
=      Z_Stop_Cmd:M20.4
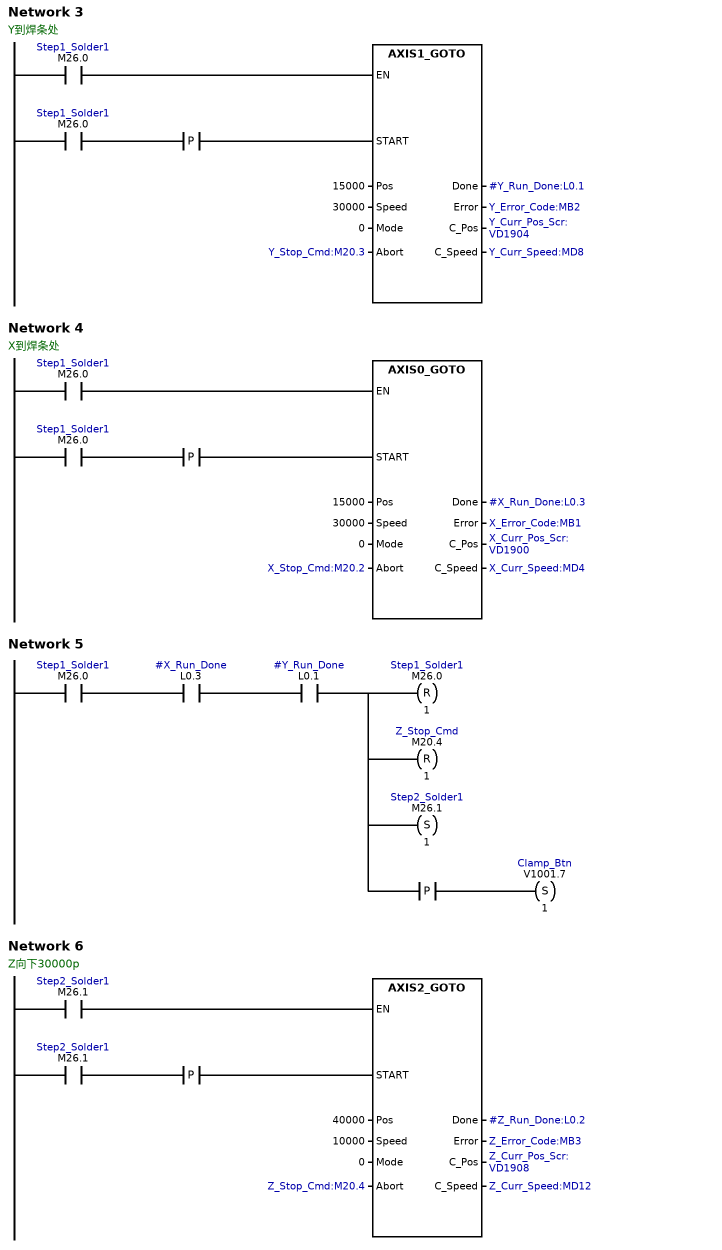
Network 3
// Y到焊条处
LD     Step1_Solder1:M26.0
=      L60.0
LD     Step1_Solder1:M26.0
EU
=      L63.7
LD     L60.0
CALL   AXIS1_GOTO:SBR14, L63.7, 15000, 30000, 0, Y_Stop_Cmd:M20.3, #Y_Run_Done:L0.1, Y_Error_Code:MB2, Y_Curr_Pos_Scr:VD1904, Y_Curr_Speed:MD8
Network 4
// X到焊条处
LD     Step1_Solder1:M26.0
=      L60.0
LD     Step1_Solder1:M26.0
EU
=      L63.7
LD     L60.0
CALL   AXIS0_GOTO:SBR3, L63.7, 15000, 30000, 0, X_Stop_Cmd:M20.2, #X_Run_Done:L0.3, X_Error_Code:MB1, X_Curr_Pos_Scr:VD1900, X_Curr_Speed:MD4
Network 5
LD     Step1_Solder1:M26.0
A      #X_Run_Done:L0.3
A      #Y_Run_Done:L0.1
R      Step1_Solder1:M26.0, 1
R      Z_Stop_Cmd:M20.4, 1
S      Step2_Solder1:M26.1, 1
EU
S      Clamp_Btn:V1001.7, 1
Network 6
// Z向下30000p
LD     Step2_Solder1:M26.1
=      L60.0
LD     Step2_Solder1:M26.1
EU
=      L63.7
LD     L60.0
CALL   AXIS2_GOTO:SBR25, L63.7, 40000, 10000, 0, Z_Stop_Cmd:M20.4, #Z_Run_Done:L0.2, Z_Error_Code:MB3, Z_Curr_Pos_Scr:VD1908, Z_Curr_Speed:MD12
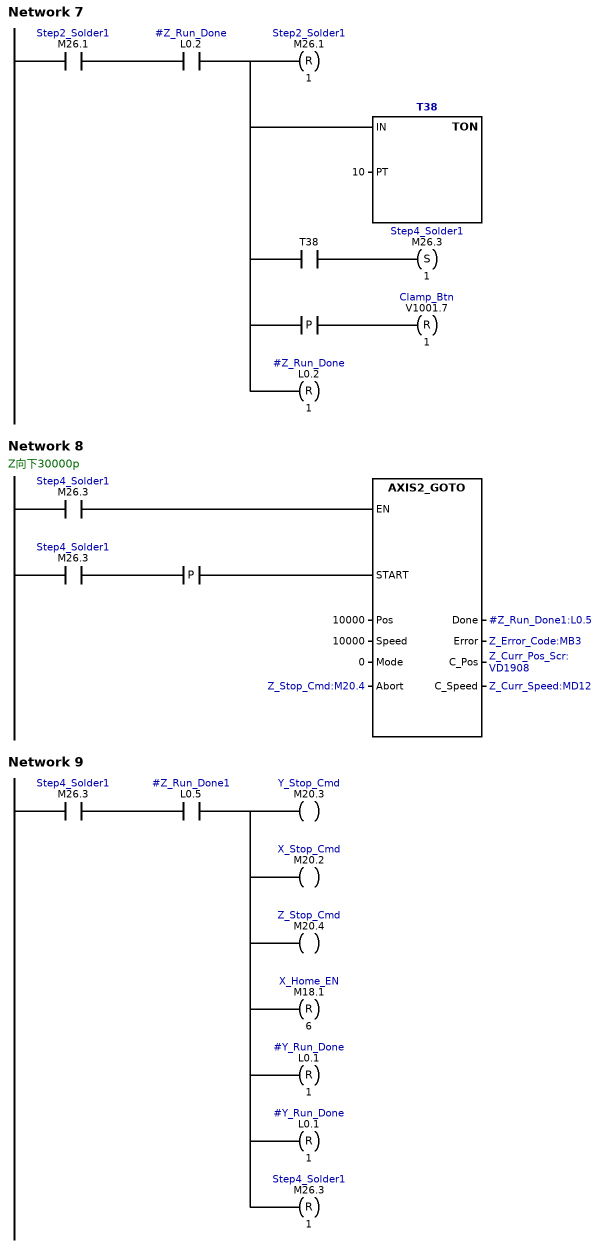
Network 7
LD     Step2_Solder1:M26.1
A      #Z_Run_Done:L0.2
LPS
R      Step2_Solder1:M26.1, 1
TON    T38, 10
A      T38
S      Step4_Solder1:M26.3, 1
LRD
EU
R      Clamp_Btn:V1001.7, 1
LPP
R      #Z_Run_Done:L0.2, 1
Network 8
// Z向下30000p
LD     Step4_Solder1:M26.3
=      L60.0
LD     Step4_Solder1:M26.3
EU
=      L63.7
LD     L60.0
CALL   AXIS2_GOTO:SBR25, L63.7, 10000, 10000, 0, Z_Stop_Cmd:M20.4, #Z_Run_Done1:L0.5, Z_Error_Code:MB3, Z_Curr_Pos_Scr:VD1908, Z_Curr_Speed:MD12
Network 9
LD     Step4_Solder1:M26.3
A      #Z_Run_Done1:L0.5
=      Y_Stop_Cmd:M20.3
=      X_Stop_Cmd:M20.2
=      Z_Stop_Cmd:M20.4
R      X_Home_EN:M18.1, 6
R      #Y_Run_Done:L0.1, 1
R      #Y_Run_Done:L0.1, 1
R      Step4_Solder1:M26.3, 1
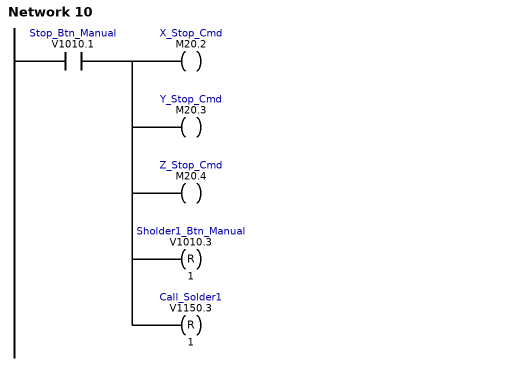
Network 10
LD     Stop_Btn_Manual:V1010.1
=      X_Stop_Cmd:M20.2
=      Y_Stop_Cmd:M20.3
=      Z_Stop_Cmd:M20.4
R      Sholder1_Btn_Manual:V1010.3, 1
R      Call_Solder1:V1150.3, 1
END_SUBROUTINE_BLOCK

SUBROUTINE_BLOCK solder2:SBR39
TITLE=子例程注释
VAR_IN_OUT
Solder2_Cmd:BOOL;	// L0.0 
END_VAR
VAR
Y_Run_Done:BOOL;	// L0.1 
Z_Run_Done:BOOL;	// L0.2 
Z_Run_Done2:BOOL;	// L0.3 
Z_Run_Done3:BOOL;	// L0.4 
Z_Run_Done1:BOOL;	// L0.5 
Z_Up_Done:BOOL;	// L0.6 
X_Run_Done1:BOOL;	// L0.7 
X_Run_Done:BOOL;	// L1.0 
Y_Run_Done1:BOOL;	// L1.1 
Y_Run_Done3:BOOL;	// L1.2 
Y_Run_Done2:BOOL;	// L1.3 
END_VAR
BEGIN
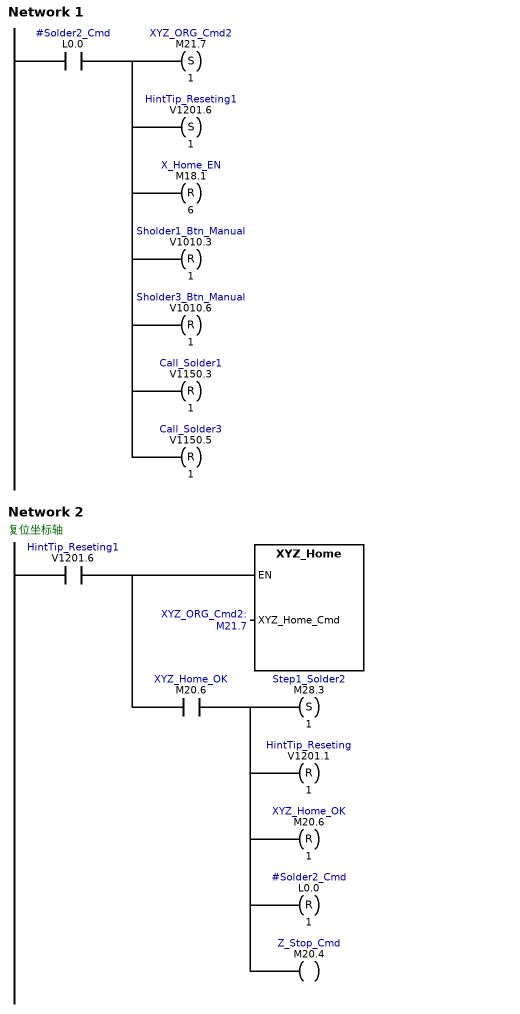
Network 1
LD     #Solder2_Cmd:L0.0
S      XYZ_ORG_Cmd2:M21.7, 1
S      HintTip_Reseting1:V1201.6, 1
R      X_Home_EN:M18.1, 6
R      Sholder1_Btn_Manual:V1010.3, 1
R      Sholder3_Btn_Manual:V1010.6, 1
R      Call_Solder1:V1150.3, 1
R      Call_Solder3:V1150.5, 1
Network 2
// 复位坐标轴
LD     HintTip_Reseting1:V1201.6
CALL   XYZ_Home:SBR37, XYZ_ORG_Cmd2:M21.7
A      XYZ_Home_OK:M20.6
S      Step1_Solder2:M28.3, 1
R      HintTip_Reseting:V1201.1, 1
R      XYZ_Home_OK:M20.6, 1
R      #Solder2_Cmd:L0.0, 1
=      Z_Stop_Cmd:M20.4
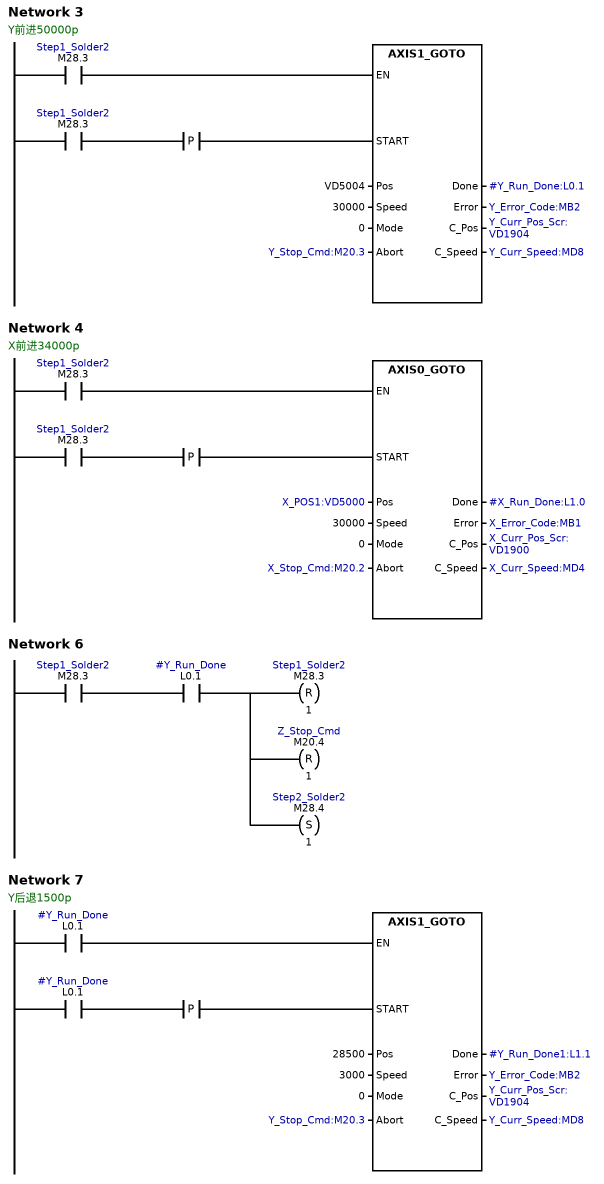
Network 3
// Y前进50000p
LD     Step1_Solder2:M28.3
=      L60.0
LD     Step1_Solder2:M28.3
EU
=      L63.7
LD     L60.0
CALL   AXIS1_GOTO:SBR14, L63.7, VD5004, 30000, 0, Y_Stop_Cmd:M20.3, #Y_Run_Done:L0.1, Y_Error_Code:MB2, Y_Curr_Pos_Scr:VD1904, Y_Curr_Speed:MD8
Network 4
// X前进34000p
LD     Step1_Solder2:M28.3
=      L60.0
LD     Step1_Solder2:M28.3
EU
=      L63.7
LD     L60.0
CALL   AXIS0_GOTO:SBR3, L63.7, X_POS1:VD5000, 30000, 0, X_Stop_Cmd:M20.2, #X_Run_Done:L1.0, X_Error_Code:MB1, X_Curr_Pos_Scr:VD1900, X_Curr_Speed:MD4
Network 6
LD     Step1_Solder2:M28.3
A      #Y_Run_Done:L0.1
R      Step1_Solder2:M28.3, 1
R      Z_Stop_Cmd:M20.4, 1
S      Step2_Solder2:M28.4, 1
Network 7
// Y后退1500p
LD     #Y_Run_Done:L0.1
=      L60.0
LD     #Y_Run_Done:L0.1
EU
=      L63.7
LD     L60.0
CALL   AXIS1_GOTO:SBR14, L63.7, 28500, 3000, 0, Y_Stop_Cmd:M20.3, #Y_Run_Done1:L1.1, Y_Error_Code:MB2, Y_Curr_Pos_Scr:VD1904, Y_Curr_Speed:MD8
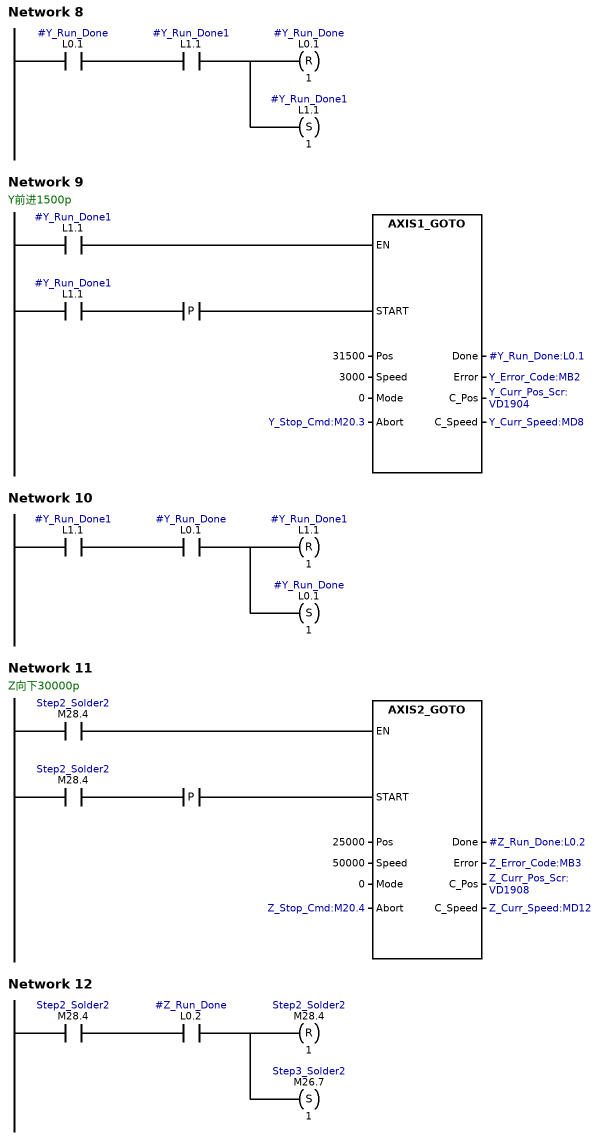
Network 8
LD     #Y_Run_Done:L0.1
A      #Y_Run_Done1:L1.1
R      #Y_Run_Done:L0.1, 1
S      #Y_Run_Done1:L1.1, 1
Network 9
// Y前进1500p
LD     #Y_Run_Done1:L1.1
=      L60.0
LD     #Y_Run_Done1:L1.1
EU
=      L63.7
LD     L60.0
CALL   AXIS1_GOTO:SBR14, L63.7, 31500, 3000, 0, Y_Stop_Cmd:M20.3, #Y_Run_Done:L0.1, Y_Error_Code:MB2, Y_Curr_Pos_Scr:VD1904, Y_Curr_Speed:MD8
Network 10
LD     #Y_Run_Done1:L1.1
A      #Y_Run_Done:L0.1
R      #Y_Run_Done1:L1.1, 1
S      #Y_Run_Done:L0.1, 1
Network 11
// Z向下30000p
LD     Step2_Solder2:M28.4
=      L60.0
LD     Step2_Solder2:M28.4
EU
=      L63.7
LD     L60.0
CALL   AXIS2_GOTO:SBR25, L63.7, 25000, 50000, 0, Z_Stop_Cmd:M20.4, #Z_Run_Done:L0.2, Z_Error_Code:MB3, Z_Curr_Pos_Scr:VD1908, Z_Curr_Speed:MD12
Network 12
LD     Step2_Solder2:M28.4
A      #Z_Run_Done:L0.2
R      Step2_Solder2:M28.4, 1
S      Step3_Solder2:M26.7, 1
